TYPE (* An Enumerated Data Type *)
  (* Standard: 61499-2 *)
  (* Version 0.0, 2003-12-06, JHC, Rockwell Automation *)
  (* Compiler header: package fb.rt.template; *)
  (* ASN.1 tag PRIVATE 6 *)
  Enumerated : (
    A, (* Enumerated value 0 *)
    B, (* Enumerated value 1 *)
    C (* Enumerated value 2 *)
  );
END_TYPE
